FUNCTION_BLOCK FB_XPIM
VAR_IN_OUT
	stYStage: DUT_MotionStage;
	stZoomStage: DUT_MotionStage;
	stFocusStage: DUT_MotionStage;
END_VAR
VAR_INPUT
	fPolished: LREAL;
	fFrosted: LREAL;
	fReticle: LREAL;
	fOut: LREAL;
END_VAR
VAR
	fbYStage: FB_MotionStage;
	fbZoom: FB_MotionStage;
	fbFocus: FB_MotionStage;
	
	{attribute 'pytmc' := '
		pv: STATES
		io: io
	'}
	fbStates: FB_XPIM_States;
	
	{attribute 'pytmc' := '
		pv: MFW
	'}
	fbFilterWheel: FB_XPIM_FilterWheel;
	
	{attribute 'pytmc' := '
		pv: CAM
	'}
	fbOpal: FB_XPIM_Opal;
	
	{attribute 'pytmc' := '
		pv: SFW
	'}
	fbFlowSwitch: FB_XTES_Flowswitch;
END_VAR

fbYStage(stMotionStage:=stYStage);
fbStates(
	stMotionStage:=stYStage,
	fPolished:=fPolished,
	fFrosted:=fFrosted,
	fReticle:=fReticle,
	fOut:=fOut);
fbZoom(stMotionStage:=stZoomStage);
fbFocus(stMotionStage:=stFocusStage);
fbFilterWheel(bExecute:=TRUE);
fbOpal();
fbFlowSwitch();

END_FUNCTION_BLOCK

(* stored: Version 1.1.0.1, ProductVersion 3.1.4022.12
   POU FB_XPIM: Id {aa9f645d-c463-4c9e-8962-8aa3b3b2b9c3}, SpecialFunc None *)
